// Link manager
FUNCTION_BLOCK FB_LinkManager IMPLEMENTS I_LinkManager
VAR
	aLinks			: ARRAY [0..nMaxSize - 1] OF FB_Link;	// Array of links
	nSize			: INT;									// Number of links in the array
END_VAR
VAR CONSTANT
	nMaxSize		: INT := 100;							// Maximum number of IOs in a group
END_VAR

// Commit link so it can be executed
METHOD CommitLink
IF nSize < nMaxSize THEN
	nSize := nSize + 1;
END_IF
END_METHOD

// Execute links
METHOD Execute
VAR
	i		: INT;		// Iterator variable
END_VAR
// Execute all links
FOR i := 0 TO nSize - 1 DO
	aLinks[i].Execute();
END_FOR
END_METHOD

METHOD GetLink : I_Link
VAR_INPUT
	nIndex		: INT;		// Link index
END_VAR
GetLink := aLinks[nIndex];
END_METHOD

// Returns a link that can be configured and then committed
PROPERTY Link : I_Link
GET
Link := aLinks[nSize];
END_GET
END_PROPERTY

END_FUNCTION_BLOCK

(* stored: Version 1.1.0.1, ProductVersion 3.1.4024.12
   POU FB_LinkManager: Id {a192d699-b6d1-4b1f-a60b-ed76d0a612c7}, SpecialFunc None
   Folder Methods: Id {aba4ef6c-931d-4c83-a958-576d5433ae95}
   Folder Properties: Id {25d22b82-de27-49e5-b7ae-24a2acc0ee71}
   Method CommitLink: Id {89d84ba9-5e8e-47be-abeb-0fce12dcdb68}
   Method Execute: Id {7b1d0740-15ff-46c5-912e-fdb9053862e7}
   Method GetLink: Id {2665f036-fcbf-44fc-915d-093e31eb5a2d}
   Property Link: Id {e10bf8e0-585f-481e-920e-184edc81dbf1}
   Get Get: Id {0527eadf-6df6-4f9a-98e1-3c80ae9d82ad} *)
